Xinje XCPPro project, PLC1: XC3-24 (software 3.3q)

PROGRAM Ladder

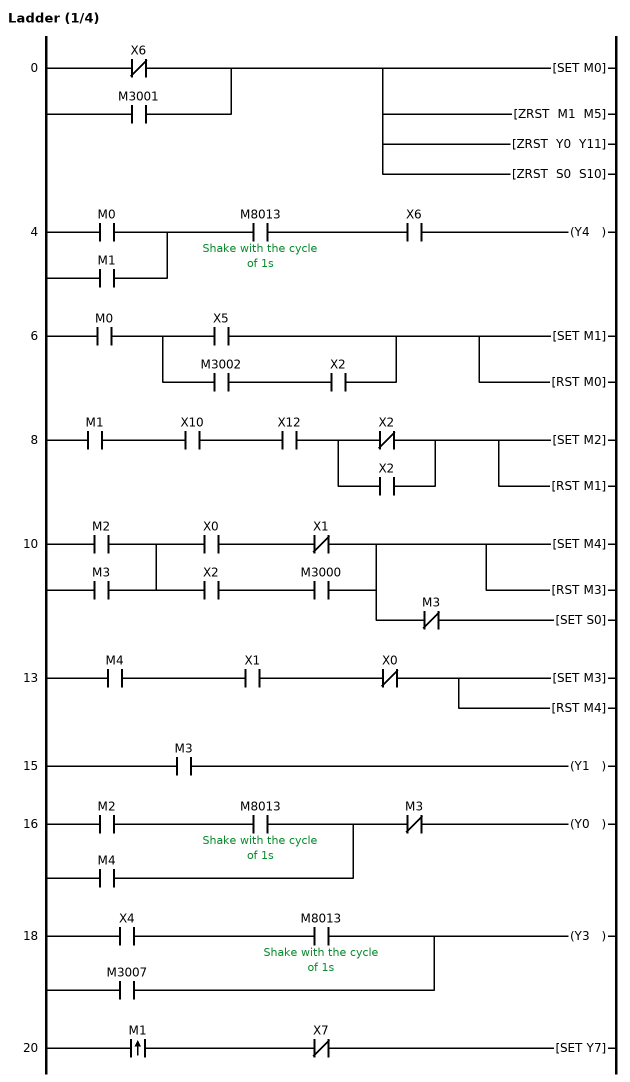
LDI    X6
OR     M3001
SET    M0
ZRST   M1 M5
ZRST   Y0 Y11
ZRST   S0 S10
LD     M0
OR     M1
AND    M8013	; Shake with the cycle of 1s
AND    X6
OUT    Y4
LD     M0
LD     X5
LD     M3002
AND    X2
ORB
ANB
SET    M1
RST    M0
LD     M1
AND    X10
AND    X12
LDI    X2
OR     X2
ANB
SET    M2
RST    M1
LD     M2
OR     M3
LD     X0
ANI    X1
LD     X2
AND    M3000
ORB
ANB
SET    M4
RST    M3
ANI    M3
SET    S0
LD     M4
AND    X1
ANI    X0
SET    M3
RST    M4
LD     M3
OUT    Y1
LD     M2
AND    M8013	; Shake with the cycle of 1s
OR     M4
ANI    M3
OUT    Y0
LD     X4
AND    M8013	; Shake with the cycle of 1s
OR     M3007
OUT    Y3
LDP    M1
ANI    X7
SET    Y7

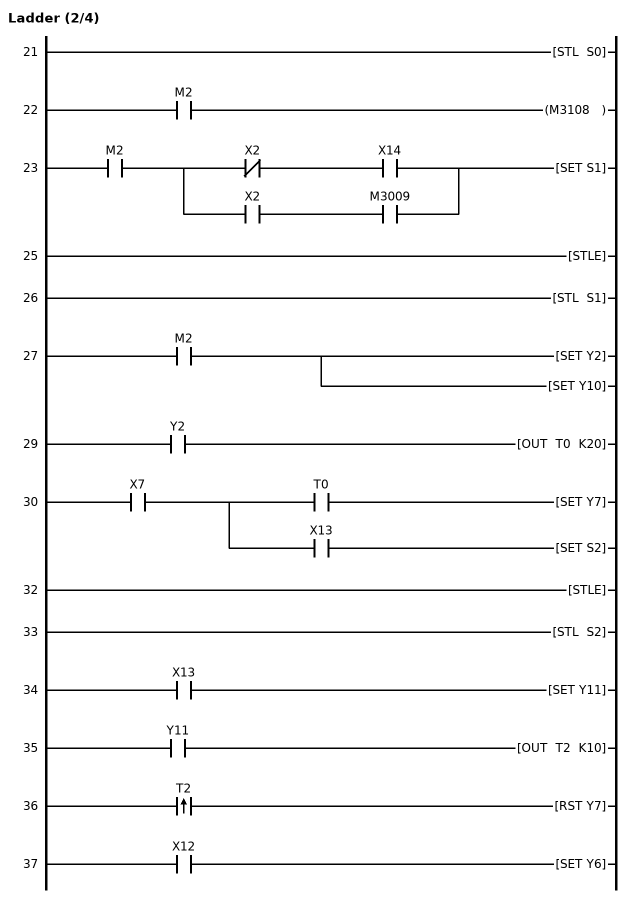
STL    S0
LD     M2
OUT    M3108
LD     M2
LDI    X2
AND    X14
LD     X2
AND    M3009
ORB
ANB
SET    S1
STLE
STL    S1
LD     M2
SET    Y2
SET    Y10
LD     Y2
OUT    T0 K20
LD     X7
MPS
AND    T0
SET    Y7
MPP
AND    X13
SET    S2
STLE
STL    S2
LD     X13
SET    Y11
LD     Y11
OUT    T2 K10
LDP    T2
RST    Y7
LD     X12
SET    Y6

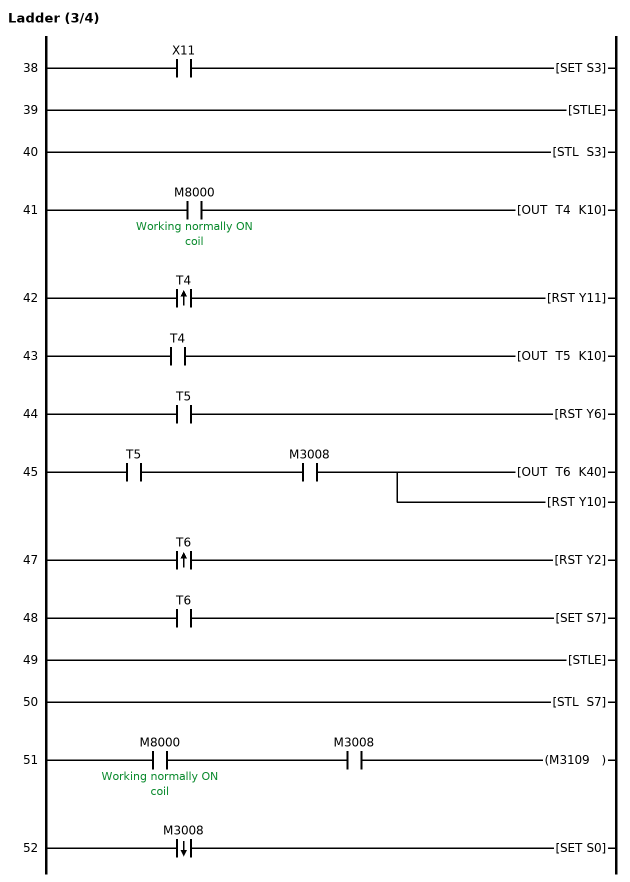
LD     X11
SET    S3
STLE
STL    S3
LD     M8000	; Working normally ON coil
OUT    T4 K10
LDP    T4
RST    Y11
LD     T4
OUT    T5 K10
LD     T5
RST    Y6
LD     T5
AND    M3008
OUT    T6 K40
RST    Y10
LDP    T6
RST    Y2
LD     T6
SET    S7
STLE
STL    S7
LD     M8000	; Working normally ON coil
AND    M3008
OUT    M3109
LDF    M3008
SET    S0

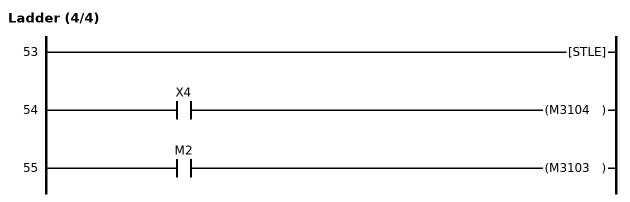
STLE
LD     X4
OUT    M3104
LD     M2
OUT    M3103